Staubli VAL3: encoder.pgx

program encoder()
  local bool l_bRisenEdge
  local bool l_bTriggerAck
  local num l_nTriggerCount
begin
  // This routine manages the encoder input of the stäubli STARC board
  //
  //
  //----------------------------------------------------------------
  //
  l_bTriggerAck=true
  l_nTriggerCount=0
  do
    // Read current encoder position
    nEncValue=aioGet(aiEncCurrentPos)
    //
    // Re-enable the latch feature of the encoder input on Stäubli STARC board
    //   if latching enabled by the conveyor library, and
    //   if there isn't a part being detected
    if (bLatchEnabled==true) and (diLatchSignal==!bLatchLevel)
      if doEnableLatch==false and l_bTriggerAck==true
        // Enable latch. (The output will be set automatically to off after latching)
        doEnableLatch=true
        l_bTriggerAck=false
      endIf
    endIf
    //
    // Check if latch feature is enabled by conveyor library
    if bLatchEnabled==true
      // check for rising edge on the Latch Input
      call _DetectIOEdge((diEncLatched==true),bMemoLatchState,l_bRisenEdge)
      //
      if l_bRisenEdge==true
        // Check number of latch for part detection
        l_nTriggerCount=l_nTriggerCount+1
        l_bTriggerAck=true
        if l_nTriggerCount>=nLatchPeriod
          // Compute Latched value
          nEncLatchedVal=aioGet(aiEncLatchedPos)
          bPartLatched=true
          l_nTriggerCount=0
        endIf
      endIf
    endIf
    //
    // ***** RESET SECTION
    if bReset
      doResetErr=true
      nEncLatchedVal=nEncValue=0
      l_nTriggerCount=0
      bReset=false
    endIf
    delay(0)
  until false
end
